TEXTLIST TextList_Navigation
  0 = 'Syn pomp' | FR: 'Synoptique\nPompage' | EN: 'Pumping\nSynoptic'
  1 = 'Syn proc' | FR: 'Synoptique\nProcédé' | EN: 'Process\nSynoptic'
  2 = 'SA'
  3 = 'Conf pomp' | FR: 'Pompage' | EN: 'Pumping'
  4 = 'Conf evap' | FR: 'Evaporation' | EN: 'Evaporation'
  5 = 'Conf mvts' | FR: 'Mouvements' | EN: 'Movements'
  6 = 'sa pomp ch' | FR: 'Pompage chambre' | EN: 'Chamber pumping'
  7 = 'sa pomp sas' | FR: 'Pompage sas' | EN: 'Loadlock pumping'
  8 = 'Conf gaz\t' | FR: 'Gaz' | EN: 'Gas'
  9 = 'Conf IAD' | FR: 'IAD' | EN: 'IAD'
  10 = 'Conf Chauf' | FR: 'Chauffage' | EN: 'Heating'
  11 = 'Effluvage' | FR: 'Effluvage' | EN: 'Glow discharge'
  12 = 'Conf Serv' | FR: 'Servitudes' | EN: 'Easements'
  13 = 'Cryo' | FR: 'Cryo' | EN: 'Cryo'
   = ''
END_TEXTLIST

(* stored: Version 1.1.0.1, ProductVersion 3.1.4026.18
   TextList TextList_Navigation: Id {c226c0a9-96ce-4186-b78d-b2b4a426ad0d} *)
